Staubli VAL3: stop.pgx

program stop()
begin

  while true




    delay(0)
  endWhile






end
